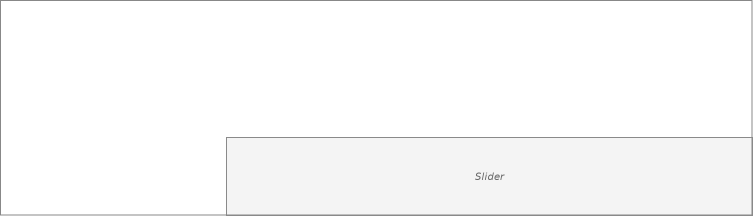
VISUALIZATION Visualization  // 753x216
    Slider (226,137 527x79), variable: MAIN.ValveOpeningControl, scale 0..1
END_VISUALIZATION

(* stored: Version 1.1.0.1, ProductVersion 3.1.4024.9
   Visu Visualization: Id {d8dee94c-064f-4243-8341-9a26801948ea} *)
